// TIA Portal V19 export
FUNCTION_BLOCK "FmStsCodes"   // FB2, LAD
{ S7_Optimized_Access := 'TRUE' }
// stored: MemoryReserve 100, SetENOAutomatically false
   VAR_INPUT
      StsIn : Byte;
   END_VAR
   VAR_OUTPUT
      "Maint alarm" : Bool;
      "Process Issue" : Bool;
      "Function Check" : Bool;
      "Uncertain Initial val" : Bool;
      "Uncertain Maint demand" : Bool;
      "Uncertain Process Related" : Bool;
      Ok : Bool;
      "OK maint advised" : Bool;
      "OK function Check" : Bool;
   END_VAR
   VAR
      Val1 : Byte;
   END_VAR
BEGIN

REGION Network 1: 0x24 = 36 BAD maintenance alarm
   // A measured value is not available because a device
   // error has occurred
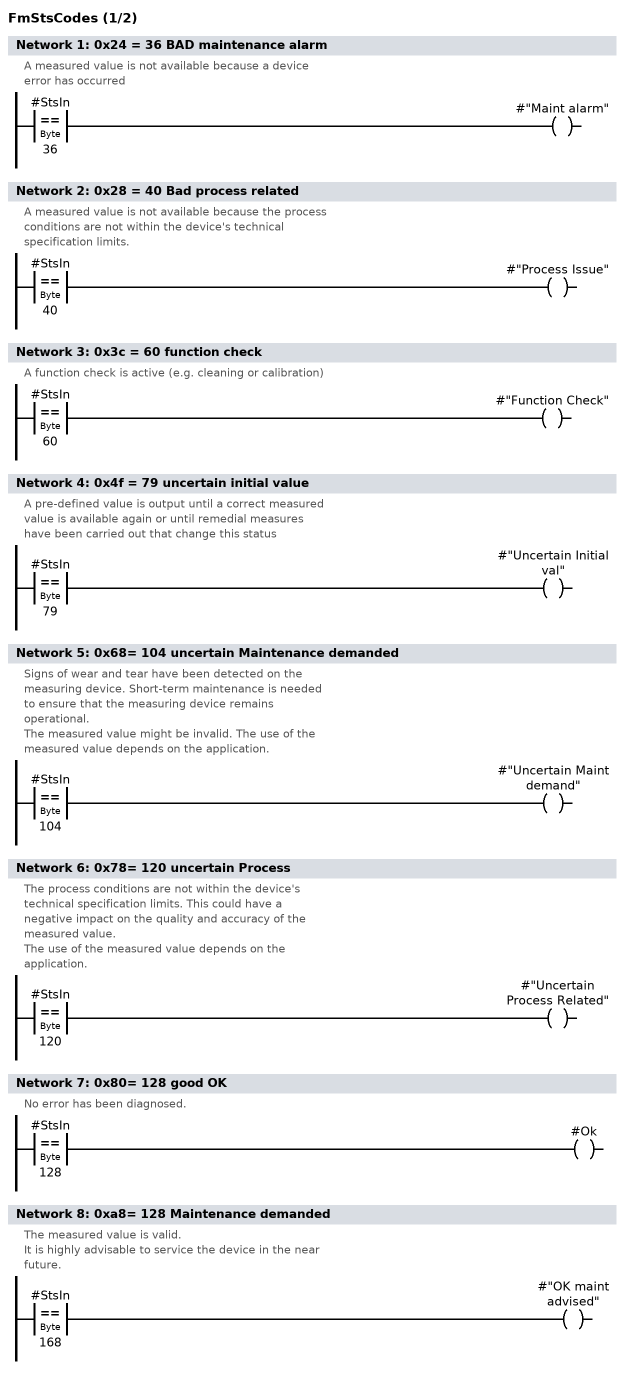
   RUNG wire#powerrail
      { S7_Templates := "SrcType := Byte" } EQ_Contact(in1 := #StsIn, in2 := 36)
      Coil( #"Maint alarm" )
   END_RUNG
   // the same network as SCL:
   #"Maint alarm" := #StsIn = 36;
END_REGION

REGION Network 2: 0x28 = 40 Bad process related
   // A measured value is not available because the process
   // conditions are not within the device's technical
   // specification limits.
   RUNG wire#powerrail
      { S7_Templates := "SrcType := Byte" } EQ_Contact(in1 := #StsIn, in2 := 40)
      Coil( #"Process Issue" )
   END_RUNG
   // the same network as SCL:
   #"Process Issue" := #StsIn = 40;
END_REGION

REGION Network 3: 0x3c = 60 function check
   // A function check is active (e.g. cleaning or calibration)
   RUNG wire#powerrail
      { S7_Templates := "SrcType := Byte" } EQ_Contact(in1 := #StsIn, in2 := 60)
      Coil( #"Function Check" )
   END_RUNG
   // the same network as SCL:
   #"Function Check" := #StsIn = 60;
END_REGION

REGION Network 4: 0x4f = 79 uncertain initial value
   // A pre-defined value is output until a correct measured
   // value is available again or until remedial measures
   // have been carried out that change this status
   RUNG wire#powerrail
      { S7_Templates := "SrcType := Byte" } EQ_Contact(in1 := #StsIn, in2 := 79)
      Coil( #"Uncertain Initial val" )
   END_RUNG
   // the same network as SCL:
   #"Uncertain Initial val" := #StsIn = 79;
END_REGION

REGION Network 5: 0x68= 104 uncertain Maintenance demanded
   // Signs of wear and tear have been detected on the
   // measuring device. Short-term maintenance is needed
   // to ensure that the measuring device remains
   // operational.
   // The measured value might be invalid. The use of the
   // measured value depends on the application.
   RUNG wire#powerrail
      { S7_Templates := "SrcType := Byte" } EQ_Contact(in1 := #StsIn, in2 := 104)
      Coil( #"Uncertain Maint demand" )
   END_RUNG
   // the same network as SCL:
   #"Uncertain Maint demand" := #StsIn = 104;
END_REGION

REGION Network 6: 0x78= 120 uncertain Process
   // The process conditions are not within the device's
   // technical specification limits. This could have a
   // negative impact on the quality and accuracy of the
   // measured value.
   // The use of the measured value depends on the
   // application.
   RUNG wire#powerrail
      { S7_Templates := "SrcType := Byte" } EQ_Contact(in1 := #StsIn, in2 := 120)
      Coil( #"Uncertain Process Related" )
   END_RUNG
   // the same network as SCL:
   #"Uncertain Process Related" := #StsIn = 120;
END_REGION

REGION Network 7: 0x80= 128 good OK
   // No error has been diagnosed.
   RUNG wire#powerrail
      { S7_Templates := "SrcType := Byte" } EQ_Contact(in1 := #StsIn, in2 := 128)
      Coil( #Ok )
   END_RUNG
   // the same network as SCL:
   #Ok := #StsIn = 128;
END_REGION

REGION Network 8: 0xa8= 128 Maintenance demanded
   // The measured value is valid.
   // It is highly advisable to service the device in the near
   // future.
   RUNG wire#powerrail
      { S7_Templates := "SrcType := Byte" } EQ_Contact(in1 := #StsIn, in2 := 168)
      Coil( #"OK maint advised" )
   END_RUNG
   // the same network as SCL:
   #"OK maint advised" := #StsIn = 168;
END_REGION

REGION Network 9: 0xbc= 188 GOOD - Function check
   // The measured value is valid.
   // The measuring device is performing an internal
   // function check. The function check does not have any
   // noticeable effect on the process.
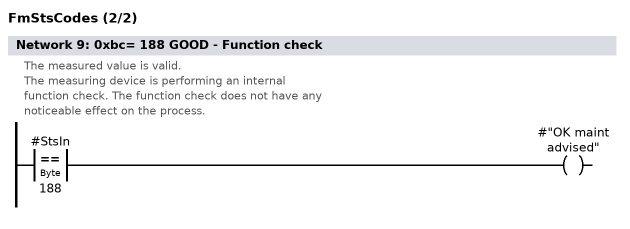
   RUNG wire#powerrail
      { S7_Templates := "SrcType := Byte" } EQ_Contact(in1 := #StsIn, in2 := 188)
      Coil( #"OK maint advised" )
   END_RUNG
   // the same network as SCL:
   #"OK maint advised" := #StsIn = 188;
END_REGION
END_FUNCTION_BLOCK
